% RSLogix 500 project AUTOMATIC_TEA_PROCESS.RSS, saved by version 8.40.00.08 %
PROJECT "UNTITLED"    % processor: MicroLogix 1200 %

PROGRAM FILES
  LAD 2   33 rungs

DATA FILES
  O0 OUTPUT  7 elements
  I1 INPUT  10 elements
  S2 STATUS  66 elements
  B3 BINARY  4 elements
  T4 TIMER  6 elements
  C5 COUNTER  1 elements
  R6 CONTROL  1 elements
  N7 INTEGER  1 elements
  F8 FLOAT  1 elements
  B23   5 elements

LADDER 2
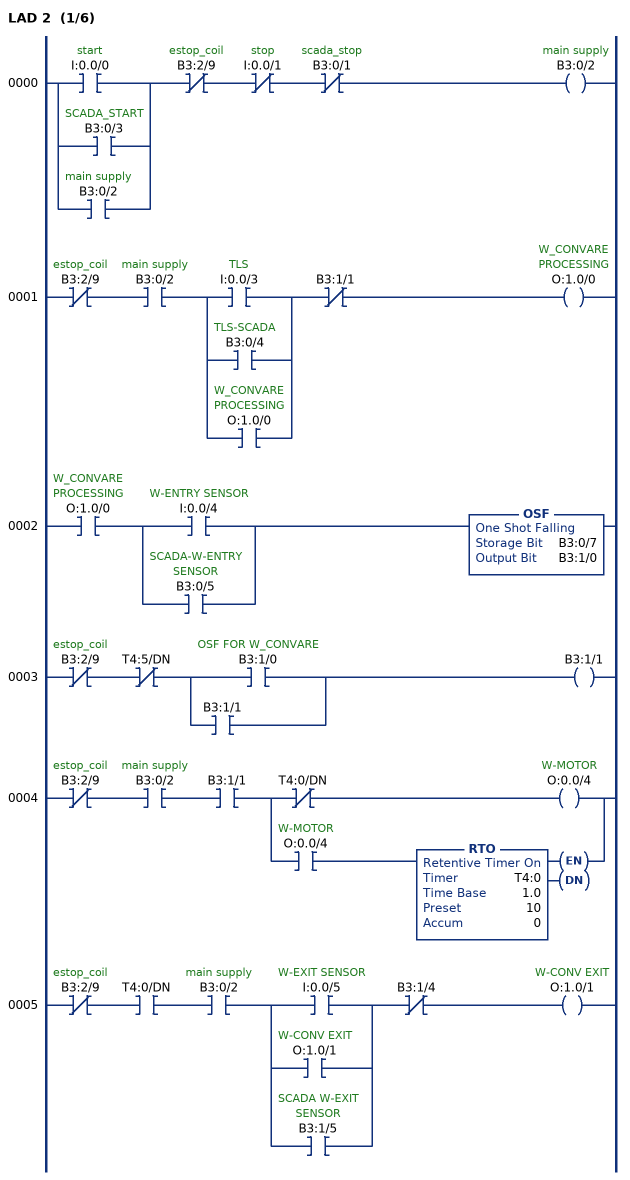
% Rung: 0 %
SOR BST XIC I:0.0/0 NXB BST XIC B3:0/3 NXB XIC B3:0/2 BND BND XIO B3:2/9 XIO I:0.0/1 XIO B3:0/1 OTE B3:0/2 EOR
%   I:0.0/0  "start" %
%   B3:0/3  "SCADA_START" %
%   B3:0/2  "main supply" %
%   B3:2/9  "estop_coil" %
%   I:0.0/1  "stop" %
%   B3:0/1  "scada_stop" %
% Rung: 1 %
SOR XIO B3:2/9 XIC B3:0/2 BST XIC I:0.0/3 NXB BST XIC B3:0/4 NXB XIC O:1.0/0 BND BND XIO B3:1/1 OTE O:1.0/0 EOR
%   B3:2/9  "estop_coil" %
%   B3:0/2  "main supply" %
%   I:0.0/3  "TLS" %
%   B3:0/4  "TLS-SCADA" %
%   O:1.0/0  "W_CONVARE PROCESSING" %
% Rung: 2 %
SOR XIC O:1.0/0 BST XIC I:0.0/4 NXB XIC B3:0/5 BND OSF B3:0/7 B3:1/0 EOR
%   O:1.0/0  "W_CONVARE PROCESSING" %
%   I:0.0/4  "W-ENTRY SENSOR" %
%   B3:0/5  "SCADA-W-ENTRY SENSOR" %
%   B3:1/0  "OSF FOR W_CONVARE" %
% Rung: 3 %
SOR XIO B3:2/9 XIO T4:5/DN BST XIC B3:1/0 NXB XIC B3:1/1 BND OTE B3:1/1 EOR
%   B3:2/9  "estop_coil" %
%   B3:1/0  "OSF FOR W_CONVARE" %
% Rung: 4 %
SOR XIO B3:2/9 XIC B3:0/2 XIC B3:1/1 BST XIO T4:0/DN OTE O:0.0/4 NXB XIC O:0.0/4 RTO T4:0 1.0 10 0 BND EOR
%   B3:2/9  "estop_coil" %
%   B3:0/2  "main supply" %
%   O:0.0/4  "W-MOTOR" %
% Rung: 5 %
SOR XIO B3:2/9 XIC T4:0/DN XIC B3:0/2 BST BST XIC I:0.0/5 NXB XIC O:1.0/1 BND NXB XIC B3:1/5 BND XIO B3:1/4 OTE O:1.0/1 EOR
%   B3:2/9  "estop_coil" %
%   B3:0/2  "main supply" %
%   I:0.0/5  "W-EXIT SENSOR" %
%   O:1.0/1  "W-CONV EXIT" %
%   B3:1/5  "SCADA W-EXIT SENSOR" %

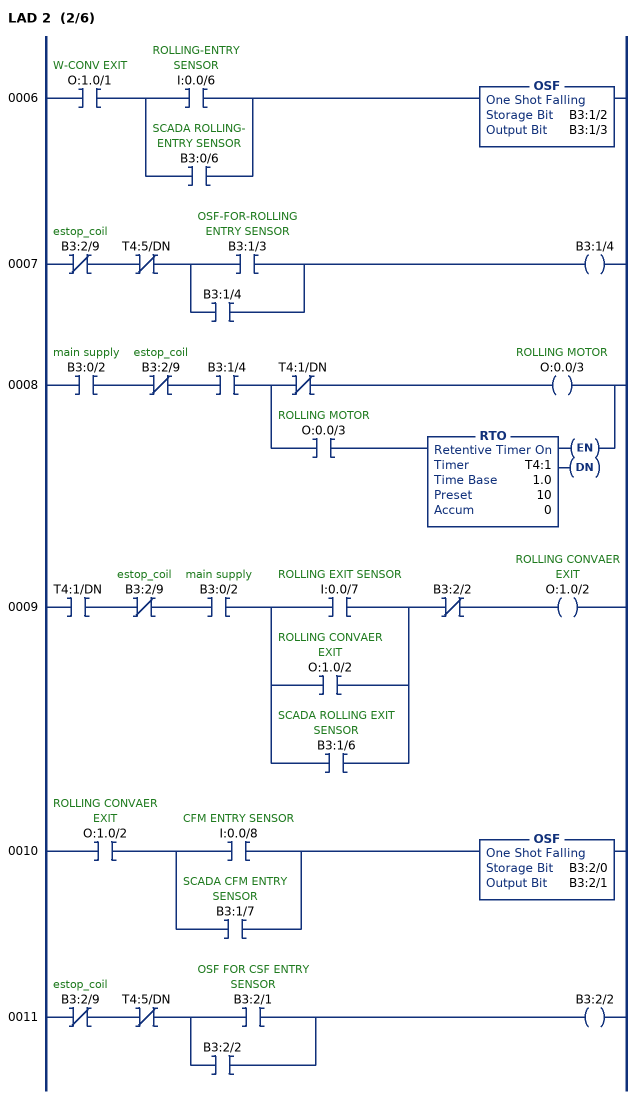
% Rung: 6 %
SOR XIC O:1.0/1 BST XIC I:0.0/6 NXB XIC B3:0/6 BND OSF B3:1/2 B3:1/3 EOR
%   O:1.0/1  "W-CONV EXIT" %
%   I:0.0/6  "ROLLING-ENTRY SENSOR" %
%   B3:0/6  "SCADA ROLLING-ENTRY SENSOR" %
%   B3:1/3  "OSF-FOR-ROLLING ENTRY SENSOR" %
% Rung: 7 %
SOR XIO B3:2/9 XIO T4:5/DN BST XIC B3:1/3 NXB XIC B3:1/4 BND OTE B3:1/4 EOR
%   B3:2/9  "estop_coil" %
%   B3:1/3  "OSF-FOR-ROLLING ENTRY SENSOR" %
% Rung: 8 %
SOR XIC B3:0/2 XIO B3:2/9 XIC B3:1/4 BST XIO T4:1/DN OTE O:0.0/3 NXB XIC O:0.0/3 RTO T4:1 1.0 10 0 BND EOR
%   B3:0/2  "main supply" %
%   B3:2/9  "estop_coil" %
%   O:0.0/3  "ROLLING MOTOR" %
% Rung: 9 %
SOR XIC T4:1/DN XIO B3:2/9 XIC B3:0/2 BST BST XIC I:0.0/7 NXB XIC O:1.0/2 BND NXB XIC B3:1/6 BND XIO B3:2/2 OTE O:1.0/2 EOR
%   B3:2/9  "estop_coil" %
%   B3:0/2  "main supply" %
%   I:0.0/7  "ROLLING EXIT SENSOR" %
%   O:1.0/2  "ROLLING CONVAER EXIT" %
%   B3:1/6  "SCADA ROLLING EXIT SENSOR" %
% Rung: 10 %
SOR XIC O:1.0/2 BST XIC I:0.0/8 NXB XIC B3:1/7 BND OSF B3:2/0 B3:2/1 EOR
%   O:1.0/2  "ROLLING CONVAER EXIT" %
%   I:0.0/8  "CFM ENTRY SENSOR" %
%   B3:1/7  "SCADA CFM ENTRY SENSOR" %
%   B3:2/1  "OSF FOR CSF ENTRY SENSOR" %
% Rung: 11 %
SOR XIO B3:2/9 XIO T4:5/DN BST XIC B3:2/1 NXB XIC B3:2/2 BND OTE B3:2/2 EOR
%   B3:2/9  "estop_coil" %
%   B3:2/1  "OSF FOR CSF ENTRY SENSOR" %

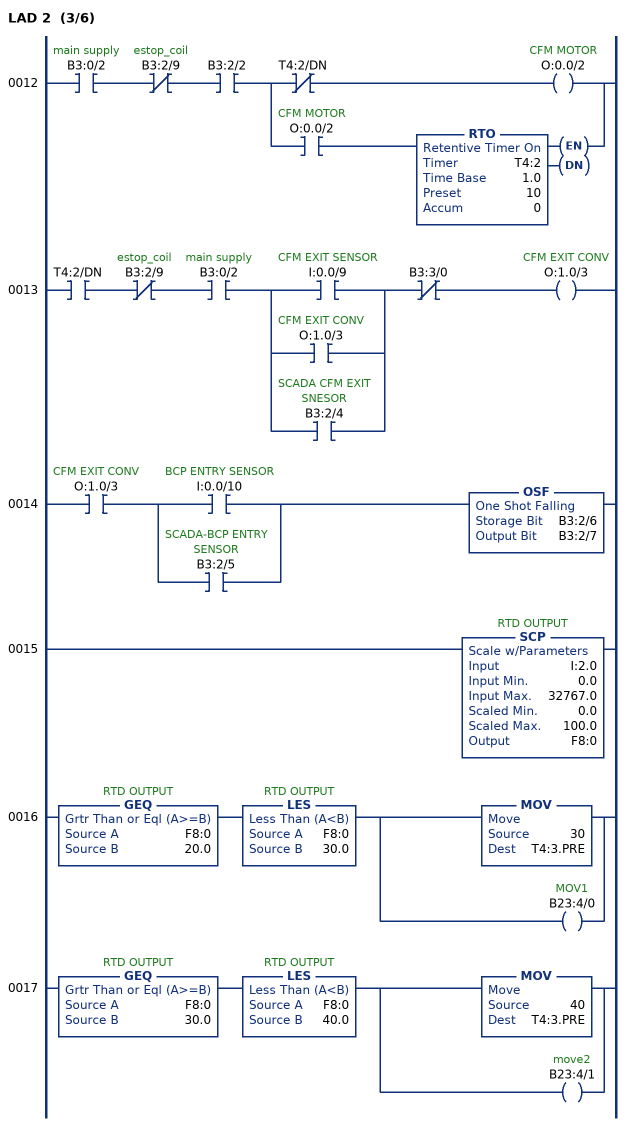
% Rung: 12 %
SOR XIC B3:0/2 XIO B3:2/9 XIC B3:2/2 BST XIO T4:2/DN OTE O:0.0/2 NXB XIC O:0.0/2 RTO T4:2 1.0 10 0 BND EOR
%   B3:0/2  "main supply" %
%   B3:2/9  "estop_coil" %
%   O:0.0/2  "CFM MOTOR" %
% Rung: 13 %
SOR XIC T4:2/DN XIO B3:2/9 XIC B3:0/2 BST BST XIC I:0.0/9 NXB XIC O:1.0/3 BND NXB XIC B3:2/4 BND XIO B3:3/0 OTE O:1.0/3 EOR
%   B3:2/9  "estop_coil" %
%   B3:0/2  "main supply" %
%   I:0.0/9  "CFM EXIT SENSOR" %
%   O:1.0/3  "CFM EXIT CONV" %
%   B3:2/4  "SCADA CFM EXIT SNESOR" %
% Rung: 14 %
SOR XIC O:1.0/3 BST XIC I:0.0/10 NXB XIC B3:2/5 BND OSF B3:2/6 B3:2/7 EOR
%   O:1.0/3  "CFM EXIT CONV" %
%   I:0.0/10  "BCP ENTRY SENSOR" %
%   B3:2/5  "SCADA-BCP ENTRY SENSOR" %
%   B3:2/7  "OSF FOR BCP ENTRY SENSOR" %
% Rung: 15 %
SOR SCP I:2.0 0.0 32767.0 0.0 100.0 F8:0 EOR
%   I:2.0  "RTD" %
%   F8:0  "RTD OUTPUT" %
% Rung: 16 %
SOR GEQ F8:0 20.0 LES F8:0 30.0 BST MOV 30 T4:3.PRE NXB OTE B23:4/0 BND EOR
%   F8:0  "RTD OUTPUT" %
%   B23:4/0  "MOV1" %
% Rung: 17 %
SOR GEQ F8:0 30.0 LES F8:0 40.0 BST MOV 40 T4:3.PRE NXB OTE B23:4/1 BND EOR
%   F8:0  "RTD OUTPUT" %
%   B23:4/1  "move2" %

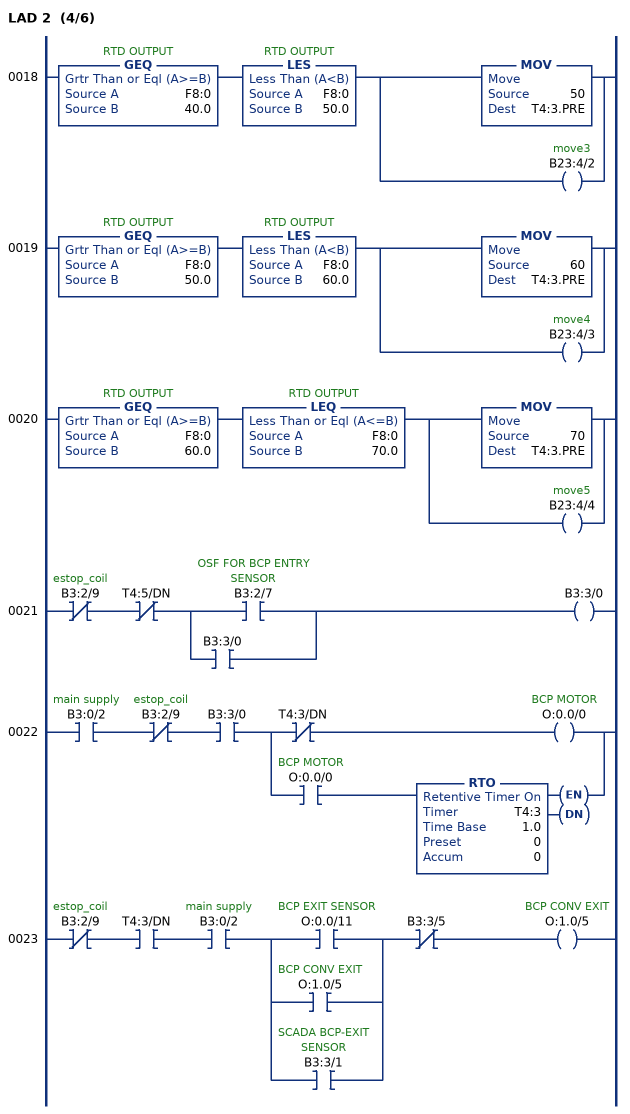
% Rung: 18 %
SOR GEQ F8:0 40.0 LES F8:0 50.0 BST MOV 50 T4:3.PRE NXB OTE B23:4/2 BND EOR
%   F8:0  "RTD OUTPUT" %
%   B23:4/2  "move3" %
% Rung: 19 %
SOR GEQ F8:0 50.0 LES F8:0 60.0 BST MOV 60 T4:3.PRE NXB OTE B23:4/3 BND EOR
%   F8:0  "RTD OUTPUT" %
%   B23:4/3  "move4" %
% Rung: 20 %
SOR GEQ F8:0 60.0 LEQ F8:0 70.0 BST MOV 70 T4:3.PRE NXB OTE B23:4/4 BND EOR
%   F8:0  "RTD OUTPUT" %
%   B23:4/4  "move5" %
% Rung: 21 %
SOR XIO B3:2/9 XIO T4:5/DN BST XIC B3:2/7 NXB XIC B3:3/0 BND OTE B3:3/0 EOR
%   B3:2/9  "estop_coil" %
%   B3:2/7  "OSF FOR BCP ENTRY SENSOR" %
% Rung: 22 %
SOR XIC B3:0/2 XIO B3:2/9 XIC B3:3/0 BST XIO T4:3/DN OTE O:0.0/0 NXB XIC O:0.0/0 RTO T4:3 1.0 0 0 BND EOR
%   B3:0/2  "main supply" %
%   B3:2/9  "estop_coil" %
%   O:0.0/0  "BCP MOTOR" %
% Rung: 23 %
SOR XIO B3:2/9 XIC T4:3/DN XIC B3:0/2 BST BST XIC O:0.0/11 NXB XIC O:1.0/5 BND NXB XIC B3:3/1 BND XIO B3:3/5 OTE O:1.0/5 EOR
%   B3:2/9  "estop_coil" %
%   B3:0/2  "main supply" %
%   O:0.0/11  "BCP EXIT SENSOR" %
%   O:1.0/5  "BCP CONV EXIT" %
%   B3:3/1  "SCADA BCP-EXIT SENSOR" %

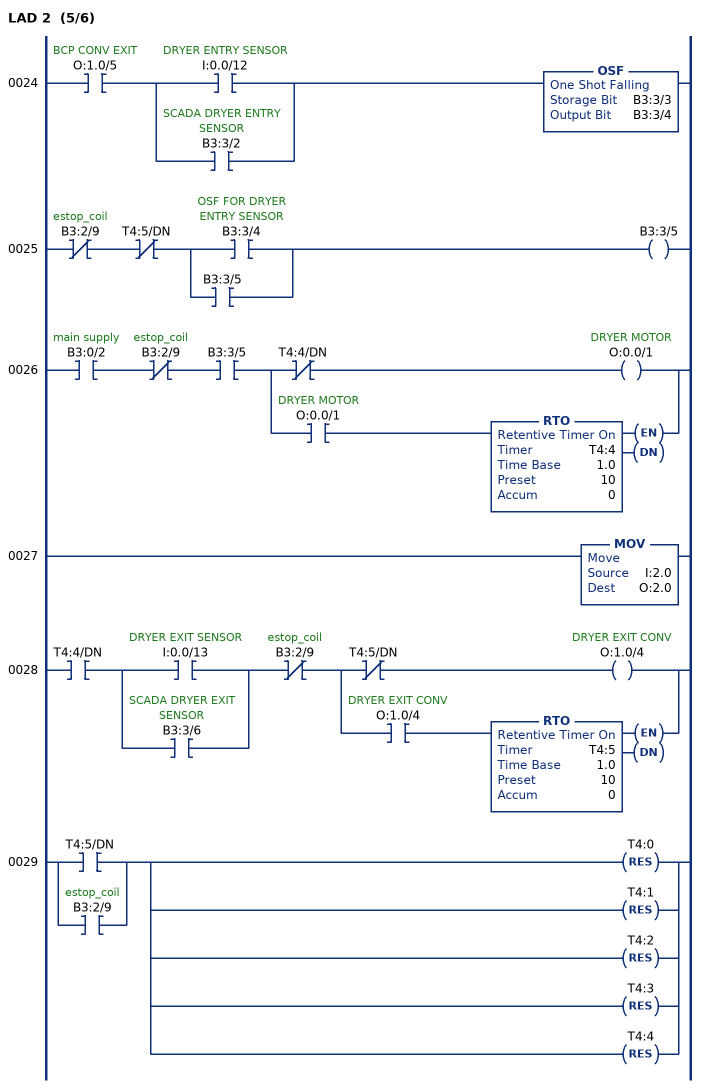
% Rung: 24 %
SOR XIC O:1.0/5 BST XIC I:0.0/12 NXB XIC B3:3/2 BND OSF B3:3/3 B3:3/4 EOR
%   O:1.0/5  "BCP CONV EXIT" %
%   I:0.0/12  "DRYER ENTRY SENSOR" %
%   B3:3/2  "SCADA DRYER ENTRY SENSOR" %
%   B3:3/4  "OSF FOR DRYER ENTRY SENSOR" %
% Rung: 25 %
SOR XIO B3:2/9 XIO T4:5/DN BST XIC B3:3/4 NXB XIC B3:3/5 BND OTE B3:3/5 EOR
%   B3:2/9  "estop_coil" %
%   B3:3/4  "OSF FOR DRYER ENTRY SENSOR" %
% Rung: 26 %
SOR XIC B3:0/2 XIO B3:2/9 XIC B3:3/5 BST XIO T4:4/DN OTE O:0.0/1 NXB XIC O:0.0/1 RTO T4:4 1.0 10 0 BND EOR
%   B3:0/2  "main supply" %
%   B3:2/9  "estop_coil" %
%   O:0.0/1  "DRYER MOTOR" %
% Rung: 27 %
SOR MOV I:2.0 O:2.0 EOR
%   I:2.0  "RTD" %
% Rung: 28 %
SOR XIC T4:4/DN BST XIC I:0.0/13 NXB XIC B3:3/6 BND XIO B3:2/9 BST XIO T4:5/DN OTE O:1.0/4 NXB XIC O:1.0/4 RTO T4:5 1.0 10 0 BND EOR
%   I:0.0/13  "DRYER EXIT SENSOR" %
%   B3:3/6  "SCADA DRYER EXIT SENSOR" %
%   B3:2/9  "estop_coil" %
%   O:1.0/4  "DRYER EXIT CONV" %
% Rung: 29 %
SOR BST XIC T4:5/DN NXB XIC B3:2/9 BND BST RES T4:0 NXB BST RES T4:1 NXB BST RES T4:2 NXB BST RES T4:3 NXB RES T4:4 BND BND BND BND EOR
%   B3:2/9  "estop_coil" %

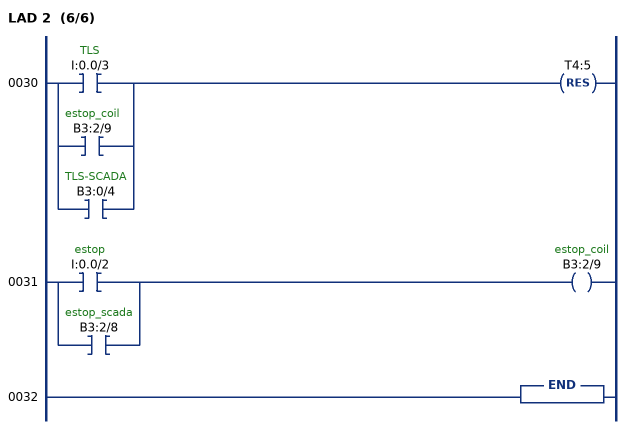
% Rung: 30 %
SOR BST BST XIC I:0.0/3 NXB XIC B3:2/9 BND NXB XIC B3:0/4 BND RES T4:5 EOR
%   I:0.0/3  "TLS" %
%   B3:2/9  "estop_coil" %
%   B3:0/4  "TLS-SCADA" %
% Rung: 31 %
SOR BST XIC I:0.0/2 NXB XIC B3:2/8 BND OTE B3:2/9 EOR
%   I:0.0/2  "estop" %
%   B3:2/8  "estop_scada" %
%   B3:2/9  "estop_coil" %
% Rung: 32 %
SOR END EOR

OTHER DOCUMENTED ADDRESSES
  B3:0/0  SCADA_START
  B3:2/3  "E-stop coil"

DATA TABLE (non-zero values as saved)
DATA T4
% .PRE .ACC %
% T4:0 % 10 0
% T4:1 % 10 0
% T4:2 % 10 0
% T4:4 % 10 0
% T4:5 % 10 0
